% RSLogix 500 project LOGIC GATE1.RSS, saved by version 8.30.00.16 %
PROJECT "UNTITLED"    % processor: Bul.1763 MicroLogix 1100 Series B %

PROGRAM FILES
  LAD 2   8 rungs

DATA FILES
  O0 OUTPUT  4 elements
  I1 INPUT  6 elements
  S2 STATUS  66 elements
  B3 BINARY  1 elements
  T4 TIMER  1 elements
  C5 COUNTER  1 elements
  R6 CONTROL  1 elements
  N7 INTEGER  1 elements
  F8 FLOAT  1 elements

LADDER 2
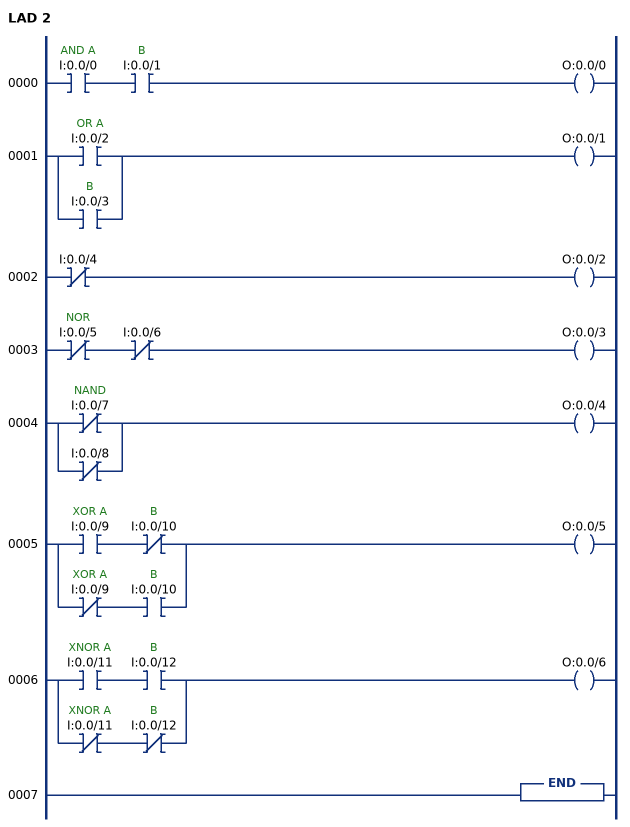
% Rung: 0 %
SOR XIC I:0.0/0 XIC I:0.0/1 OTE O:0.0/0 EOR
%   I:0.0/0  "AND A" %
%   I:0.0/1  "B" %
% Rung: 1 %
SOR BST XIC I:0.0/2 NXB XIC I:0.0/3 BND OTE O:0.0/1 EOR
%   I:0.0/2  "OR A" %
%   I:0.0/3  "B" %
% Rung: 2 %
SOR XIO I:0.0/4 OTE O:0.0/2 EOR
% Rung: 3 %
SOR XIO I:0.0/5 XIO I:0.0/6 OTE O:0.0/3 EOR
%   I:0.0/5  "NOR" %
% Rung: 4 %
SOR BST XIO I:0.0/7 NXB XIO I:0.0/8 BND OTE O:0.0/4 EOR
%   I:0.0/7  "NAND" %
% Rung: 5 %
SOR BST XIC I:0.0/9 XIO I:0.0/10 NXB XIO I:0.0/9 XIC I:0.0/10 BND OTE O:0.0/5 EOR
%   I:0.0/9  "XOR A" %
%   I:0.0/10  "B" %
% Rung: 6 %
SOR BST XIC I:0.0/11 XIC I:0.0/12 NXB XIO I:0.0/11 XIO I:0.0/12 BND OTE O:0.0/6 EOR
%   I:0.0/11  "XNOR A" %
%   I:0.0/12  "B" %
% Rung: 7 %
SOR END EOR
